
// ===== library types =====

TYPE "typeSinaSpeedInterface"
   STRUCT
      control : Struct
         enableAxis : Bool;
         ackError : Bool;
         speedSp : Real;
         refSpeed : Real;
         configAxis : Word := 16#003F;
         hwidStw : Hw_SubModule;
         hwidZsw : Hw_SubModule;
      END_STRUCT;
      status : Struct
         axisEnabled : Bool;
         lockout : Bool;
         actVelocity : Real;
         error : Bool;
         status : Int;
         diagId : Word;
      END_STRUCT;
   END_STRUCT;
END_TYPE

FUNCTION_BLOCK "SinaSpeedTest"   // FB1, LAD
{ S7_Optimized_Access := 'TRUE' }
VERSION : 0.1
   VAR_IN_OUT
      data : "typeSinaSpeedInterface";
   END_VAR
   VAR
      instSinaSpeed : SinaSpeed;
      instSinaParaS : SinaParaS;
   END_VAR
BEGIN

REGION Network 1
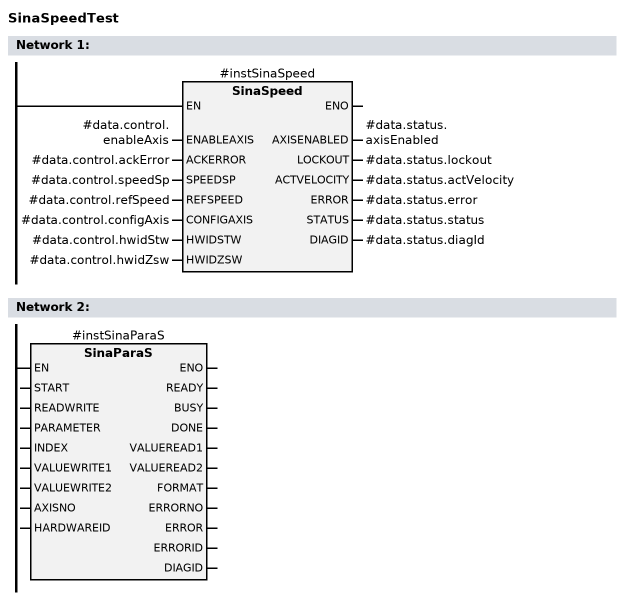
   #instSinaSpeed(EnableAxis := #data.control.enableAxis,   // SinaSpeed
                  AckError := #data.control.ackError,
                  SpeedSp := #data.control.speedSp,
                  RefSpeed := #data.control.refSpeed,
                  ConfigAxis := #data.control.configAxis,
                  HWIDSTW := #data.control.hwidStw,
                  HWIDZSW := #data.control.hwidZsw,
                  AxisEnabled => #data.status.axisEnabled,
                  Lockout => #data.status.lockout,
                  ActVelocity => #data.status.actVelocity,
                  Error => #data.status.error,
                  Status => #data.status.status,
                  DiagId => #data.status.diagId);
END_REGION

REGION Network 2
   #instSinaParaS();   // SinaParaS
END_REGION
END_FUNCTION_BLOCK

// ===== library: MasterCopy "SinaSpeedTest" =====

FUNCTION_BLOCK "SinaSpeedTest"   // FB1, LAD
{ S7_Optimized_Access := 'TRUE' }
VERSION : 0.1
   VAR_IN_OUT
      data : "typeSinaSpeedInterface";
   END_VAR
   VAR
      instSinaSpeed : SinaSpeed;
      instSinaParaS : SinaParaS;
   END_VAR
BEGIN

REGION Network 1
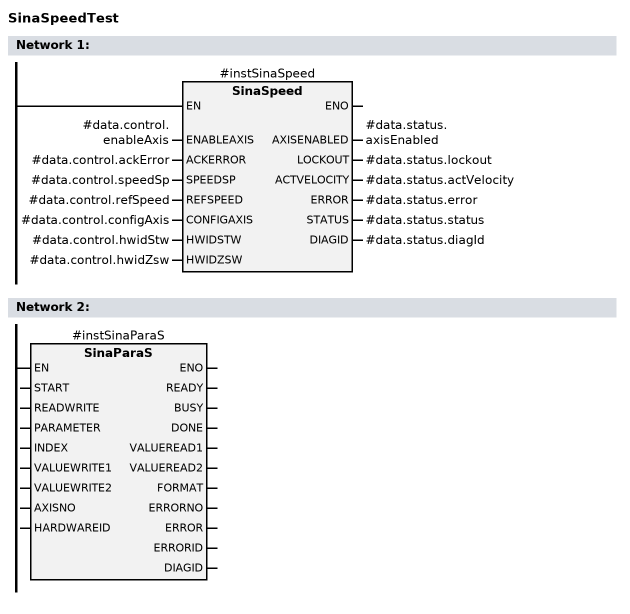
   #instSinaSpeed(EnableAxis := #data.control.enableAxis,   // SinaSpeed
                  AckError := #data.control.ackError,
                  SpeedSp := #data.control.speedSp,
                  RefSpeed := #data.control.refSpeed,
                  ConfigAxis := #data.control.configAxis,
                  HWIDSTW := #data.control.hwidStw,
                  HWIDZSW := #data.control.hwidZsw,
                  AxisEnabled => #data.status.axisEnabled,
                  Lockout => #data.status.lockout,
                  ActVelocity => #data.status.actVelocity,
                  Error => #data.status.error,
                  Status => #data.status.status,
                  DiagId => #data.status.diagId);
END_REGION

REGION Network 2
   #instSinaParaS();   // SinaParaS
END_REGION
END_FUNCTION_BLOCK